FUNCTION_BLOCK FB_TMCM1140_Rotate
VAR_INPUT
	bExecute	: BOOL;
	bStop		: BOOL;
	bCCW		: BOOL;
	nSpeed		: DINT; //Reale Einheit/s //wenn -1, dann wird ProfileSpeed genommen
END_VAR
VAR_OUTPUT
	bBusy 		: BOOL;
	bError 		: BOOL;
	nErrorId 	: ERRORID;	
END_VAR
VAR_IN_OUT
	pHwRef : POINTER TO FB_HwRefTMCM1140;
END_VAR
VAR
	nState 			: USINT;
	nCurrentSpeed 	: DINT;
	bCurrentCCW		: BOOL;	
END_VAR

IF bExecute THEN
	IF NOT pHwRef^.M_GetDS402State() = E_CoDS402States.DS402STATE_OperationEnabled THEN
		nErrorID := E_ErrorIdDS402.ERRORID_OperationNotEnabled;
		nState := 99;
	END_IF
	
	IF nState = 0 THEN
		bBusy := TRUE;
		
		IF nSpeed = -1 THEN
			nSpeed := pHwRef^.P_nMaxSpeed;
		END_IF
		
		IF NOT pHwRef^.M_SetVLSpeed(nSpeed, bCCW) THEN
			nErrorID := E_ErrorIdHwGeneral.ERRORID_InvalidSpeed;
			nState := 99;
		ELSE
			nCurrentSpeed := nSpeed;
			bCurrentCCW := bCCW;
			pHwRef^.nMode := 2;
			nState := 1;
		END_IF
		
	ELSIF nState = 1 THEN
		IF bStop THEN
			pHwRef^.M_SetVLSpeed(0, FALSE);
			nState := 2;
		ELSE
			IF nSpeed <> nCurrentSpeed OR bCCW <> bCurrentCCW THEN
				IF pHwRef^.M_SetVLSpeed(nSpeed, bCCW) THEN
					nCurrentSpeed := nSpeed;
					bCurrentCCW := bCCW;
				END_IF
			END_IF
			
		END_IF
	ELSIF nState = 2 THEN
		IF NOT pHwRef^.P_bIsMoving THEN
			nState := 80;
		END_IF
	END_IF
	
	IF nState >= 80 THEN
		bBusy := FALSE;
		IF nState = 99 THEN
			bError := TRUE;
		END_IF
	END_IF

ELSE
	bBusy := FALSE;
	bError := FALSE;
	bStop := FALSE;
	nState := 0;	
END_IF

END_FUNCTION_BLOCK

(* stored: Version 1.1.0.1, ProductVersion 3.1.4024.11
   POU FB_TMCM1140_Rotate: Id {77ba5b88-0b02-4bd4-b03d-c28e45c11b5e}, SpecialFunc None *)
